FUNCTION_BLOCK PLCOpenNullRemote IMPLEMENTS  IPLCOpenCall

METHOD Aborted : BOOL
END_METHOD

METHOD Errored : BOOL
VAR_INPUT
	ID : INT;
END_VAR
END_METHOD

METHOD Finished : BOOL
END_METHOD

{warning 'add method implementation '}
METHOD Start : BOOL
VAR_INPUT
	Command	: IPLCOpenCommand;
END_VAR
//TODO
END_METHOD

END_FUNCTION_BLOCK

(* stored: Version 1.1.0.1, ProductVersion 3.1.4024.12
   POU PLCOpenNullRemote: Id {73061230-7a8e-410b-ae26-c14eb801f0aa}, SpecialFunc None
   Method Aborted: Id {d3377050-9f4c-49f6-a051-4bcdc44d847d}
   Method Errored: Id {97c3ac24-72bd-4b21-93c4-11f805822d38}
   Method Finished: Id {6fdf66c9-5086-43d9-b213-c69b23218cc4}
   Method Start: Id {42d0f9af-461f-4d36-bb4c-e7ed19b6748a} *)
